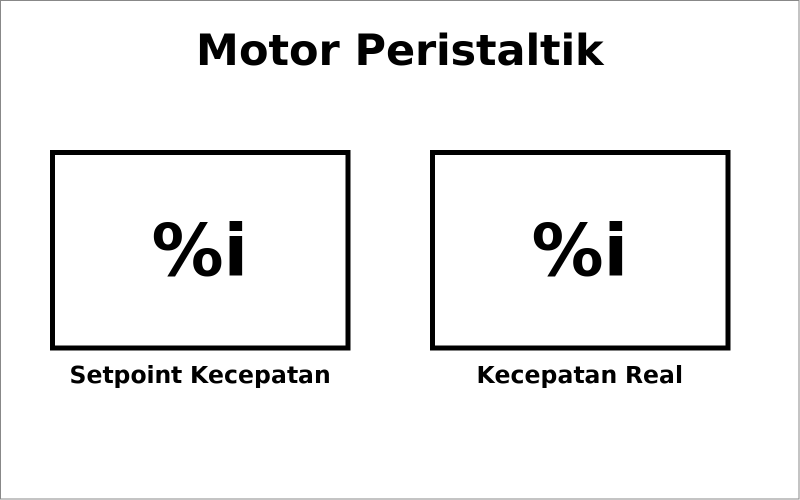
VISUALIZATION Screen_2_Sub_1  // 800x500
    Label (0,0 800x100), "Motor Peristaltik"
    Rectangle (50,150 300x200), "%i", text variable: GVL.HMI_Motor_Peristaltik_Input
        OnMouseClick: write GVL.HMI_Motor_Peristaltik_Input via VisuDialogs.Numpad
    Label (50,350 300x50), "Setpoint Kecepatan"
    Label (430,350 300x50), "Kecepatan Real"
    Rectangle (430,150 300x200), "%i", text variable: GVL.HMI_Motor_Peristaltik_Real
END_VISUALIZATION

(* stored: Version 1.1.0.1, ProductVersion 3.1.4024.12
   Visu Screen_2_Sub_1: Id {fbdae0f2-4304-4f55-9819-6741101025c2} *)
